// Mitsubishi GX Works2 project: ValueFx3uContrer3LedWTR10-E_V4   PLC: FX3U/FX3UC

PROGRAM MAIN
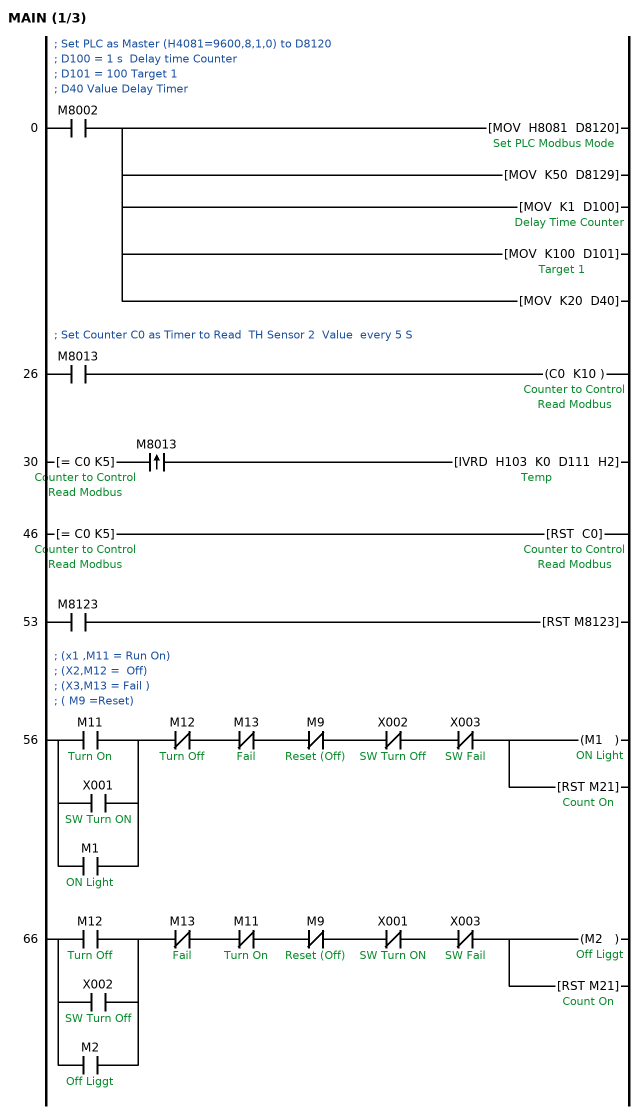
; Set PLC as Master (H4081=9600,8,1,0) to D8120
; D100 = 1 s  Delay time Counter
; D101 = 100 Target 1
; D40 Value Delay Timer
0     LD      M8002
      MOV     H8081 D8120  ; Set PLC Modbus Mode
      MOV     K50 D8129
      MOV     K1 D100  ; Delay Time Counter
      MOV     K100 D101  ; Target 1
      MOV     K20 D40
; Set Counter C0 as Timer to Read  TH Sensor 2  Value  every 5 S
26    LD      M8013
      OUT     C0 K10  ; Counter to Control Read Modbus
30    LD=     C0 K5  ; Counter to Control Read Modbus
      ANDP    M8013
      IVRD    H103 K0 D111 H2  ; Temp
46    LD=     C0 K5  ; Counter to Control Read Modbus
      RST     C0  ; Counter to Control Read Modbus
53    LD      M8123
      RST     M8123
; (x1 ,M11 = Run On)
; (X2,M12 =  Off)
; (X3,M13 = Fail )
; ( M9 =Reset)
56    LD      M11  ; Turn On
      OR      X001  ; SW Turn ON
      OR      M1  ; ON Light
      ANI     M12  ; Turn Off
      ANI     M13  ; Fail
      ANI     M9  ; Reset (Off)
      ANI     X002  ; SW Turn Off
      ANI     X003  ; SW Fail
      OUT     M1  ; ON Light
      RST     M21  ; Count On
66    LD      M12  ; Turn Off
      OR      X002  ; SW Turn Off
      OR      M2  ; Off Liggt
      ANI     M13  ; Fail
      ANI     M11  ; Turn On
      ANI     M9  ; Reset (Off)
      ANI     X001  ; SW Turn ON
      ANI     X003  ; SW Fail
      OUT     M2  ; Off Liggt
      RST     M21  ; Count On
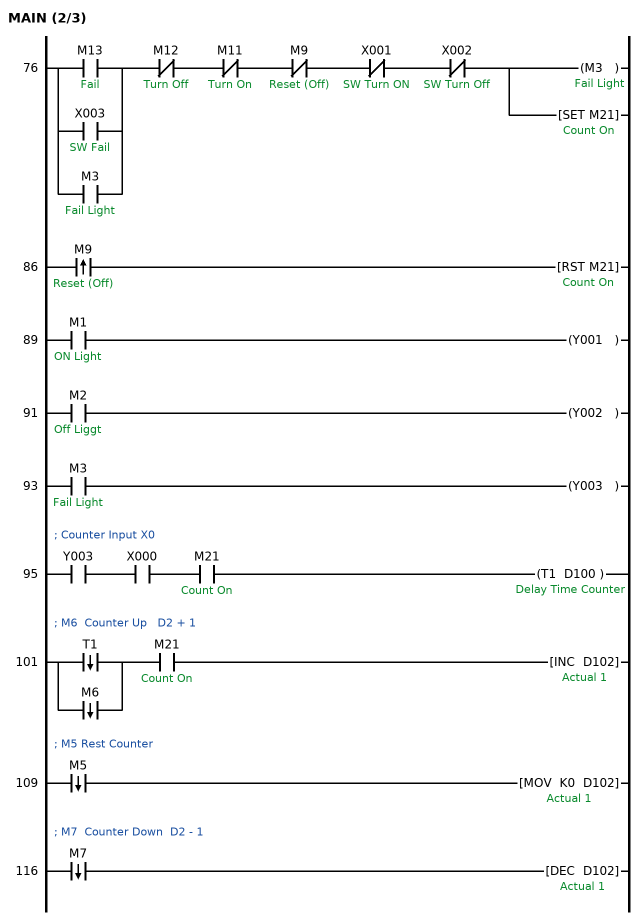
76    LD      M13  ; Fail
      OR      X003  ; SW Fail
      OR      M3  ; Fail Light
      ANI     M12  ; Turn Off
      ANI     M11  ; Turn On
      ANI     M9  ; Reset (Off)
      ANI     X001  ; SW Turn ON
      ANI     X002  ; SW Turn Off
      OUT     M3  ; Fail Light
      SET     M21  ; Count On
86    LDP     M9  ; Reset (Off)
      RST     M21  ; Count On
89    LD      M1  ; ON Light
      OUT     Y001
91    LD      M2  ; Off Liggt
      OUT     Y002
93    LD      M3  ; Fail Light
      OUT     Y003
; Counter Input X0
95    LD      Y003
      AND     X000
      AND     M21  ; Count On
      OUT     T1 D100  ; Delay Time Counter
; M6  Counter Up   D2 + 1
101   LDF     T1
      ORF     M6
      AND     M21  ; Count On
      INC     D102  ; Actual 1
; M5 Rest Counter
109   LDF     M5
      MOV     K0 D102
; M7  Counter Down  D2 - 1
116   LDF     M7
      DEC     D102
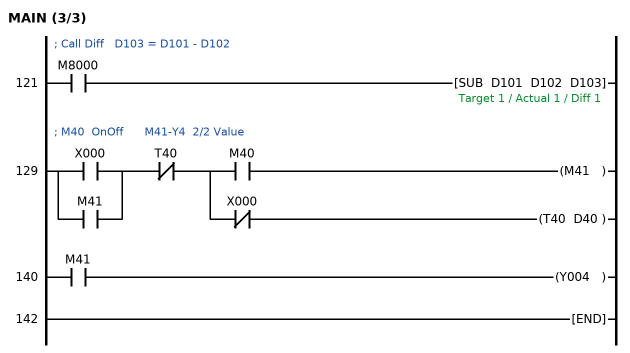
; Call Diff   D103 = D101 - D102
121   LD      M8000
      SUB     D101 D102 D103  ; Diff 1
; M40  OnOff      M41-Y4  2/2 Value
129   LD      X000
      OR      M41
      ANI     T40
      MPS
      AND     M40
      OUT     M41
      MPP
      ANI     X000
      OUT     T40 D40
140   LD      M41
      OUT     Y004
142   END
END_PROGRAM

// device comments not shown above
D112  ; Humi
D121  ; Slave No
M813  ; Reset To Read new Modbus Data
